FUNCTION_BLOCK FB_Observable_SINT EXTENDS FB_AbstractObservable
VAR
    _nVal:              SINT;
    _nOldVal:           SINT;
END_VAR

METHOD FB_init : BOOL
VAR_INPUT
    bInitRetains:       BOOL; // if TRUE, the retain variables are initialized (warm start / cold start)
    bInCopyCode:        BOOL;  // if TRUE, the instance afterwards gets moved into the copy code (online change)
END_VAR
THIS^._nTypeClass := __SYSTEM.TYPE_CLASS.TYPE_SINT;
END_METHOD

PROPERTY nDataSize : UDINT
GET
nDataSize := SIZEOF(SINT);
END_GET
END_PROPERTY

PROPERTY nValue8 : SINT
GET
nValue8 := THIS^._nVal;
END_GET
SET
THIS^._nOldVal := THIS^._nVal;
THIS^._nVal := nValue8;

THIS^.NotifyWithConditions();
END_SET
END_PROPERTY

PROPERTY PROTECTED pData : POINTER TO BYTE
GET
pData := ADR(THIS^._nVal);
END_GET
END_PROPERTY

METHOD  ValueChanged : BOOL
VAR_INPUT
END_VAR
ValueChanged := THIS^._nOldVal <> THIS^._nVal;
END_METHOD

END_FUNCTION_BLOCK

(* stored: Version 1.1.0.1, ProductVersion 3.1.4024.12
   POU FB_Observable_SINT: Id {84122a7e-3c38-05f7-368c-7f0dd6fef543}, SpecialFunc None
   Method FB_init: Id {99493679-0c61-0da6-234b-35c0c1bb959a}
   Property nDataSize: Id {54473a80-ea0a-094c-3a9c-ec97e22dca22}
   Get Get: Id {57515fb9-b273-0466-1f8d-faeb433ae9d6}
   Property nValue8: Id {a114e4fc-734c-0fe3-33a5-e563196b550c}
   Get Get: Id {96c9646f-f3d1-04ff-0a9b-cd828d7ee7f8}
   Set Set: Id {c87fc86b-5e72-0c3c-2947-5b929f4299c5}
   Property pData: Id {e2b354ad-bf44-0d5f-27fa-e55bf8e21022}
   Get Get: Id {5216bbd1-78ed-0aa4-3981-7ef4c7be7d38}
   Method ValueChanged: Id {81597bcb-d274-096a-39e2-722f7de8a406} *)
